// TIA Portal V20 export
TYPE "LKinCtrl_typePathData_PreBuf"
   STRUCT
      pathDataName : String["LKINCTRL_LENGTH_OF_PATHDATA_NAME"];   // name of PathData
      commands : Array[1.."LKINCTRL_NO_OF_PATHDATA_PREBUFFER_ELEMENTS"] of "LKinCtrl_typePathDataElement_PreBuf";   // command list
      addPointer : Int;   // pointer marking slot for adding of next command in PathDataPreBuffered
      retrievePointer : Int;   // pointer marking command entry to be read in PathDataPreBuffered
      addPointerRestarted : Bool;   // addPointer restarted after overflow
   END_STRUCT;
   // commands[1].cmdParameters.transitionParameters[1] := -1.0;
   // commands[2].cmdParameters.transitionParameters[1] := -1.0;
   // commands[3].cmdParameters.transitionParameters[1] := -1.0;
   // commands[4].cmdParameters.transitionParameters[1] := -1.0;
   // commands[5].cmdParameters.transitionParameters[1] := -1.0;
   // commands[1].parameterValid[1..4] := TRUE;
   // commands[2].parameterValid[1..4] := TRUE;
   // commands[3].parameterValid[1..4] := TRUE;
   // commands[4].parameterValid[1..4] := TRUE;
   // commands[5].parameterValid[1..4] := TRUE;
END_TYPE
